FUNCTION F_INT_RTN : INT
VAR_INPUT
	stArg : ST_Arg;
END_VAR
VAR
	sysVar_Info : __SYSTEM.VAR_INFO;
END_VAR

sysVar_Info := __VARINFO(F_INT_RTN);
IF stArg.TypeClass = sysVar_Info.TypeClass THEN 
	F_INT_RTN := TO_INT(stArg.sValue);
	END_IF

END_FUNCTION

(* stored: Version 1.1.0.1, ProductVersion 3.1.4024.4
   POU F_INT_RTN: Id {b2d50fca-2772-43a4-99b9-a237c9dab40f}, SpecialFunc None *)
